FUNCTION_BLOCK PUBLIC ABSTRACT FB_HMI_PROVIDER_BASE IMPLEMENTS ITF_HMI_PROVIDER
VAR_INPUT
END_VAR
VAR_OUTPUT
END_VAR
VAR
	eProvider	: E_HMI_PROVIDER;
	
	stItfHmiIn	: REFERENCE TO ST_HMI_IN;
	stItfHmiOut	: REFERENCE TO ST_HMI_OUT;
	
	bRequestManualControl,
	bRequestRecipeMgmt,
	bRequestSettingMgmt,
	bRequestUserMgmt,
	bMute		: BOOL;
END_VAR

PROPERTY ItfHmiIn : REFERENCE TO ST_HMI_IN
GET
ItfHmiIn REF= stItfHmiIn;
END_GET
END_PROPERTY

PROPERTY ItfHmiOut : REFERENCE TO ST_HMI_OUT
GET
ItfHmiOut REF= stItfHmiOut;
END_GET
END_PROPERTY

METHOD PUBLIC M_Init : BOOL
VAR_INPUT
END_VAR
P_HMI_Controller.M_RegisterProvider(THIS^);
M_Init := TRUE;
END_METHOD

(* reset*)
METHOD M_Reset : BOOL
stItfHmiIn.stSpecial.stButton_LedTest.bClick := FALSE;
END_METHOD

METHOD M_Run : BOOL
VAR
	msg : STRING;
END_VAR
IF NOT RefsValid THEN
	msg := CONCAT('HMI provider ref error, provider: ', TO_STRING(eProvider));
	Services.fbEventHandler.Select(TC_Events.SystemEventClass.ErrorEvent).ArgSetString(msg).Raise();
	RETURN;
END_IF

M_Run := TRUE;
END_METHOD

METHOD M_SetReferencesBase : BOOL
VAR_IN_OUT
	stHmiPrvIn	: ST_HMI_IN;
	stHmiPrvOut	: ST_HMI_OUT;
END_VAR
stItfHmiIn REF= stHmiPrvIn;
stItfHmiOut REF= stHmiPrvOut;
stItfHmiOut.stCommon REF= HMI.stHmi.stOut.stCommon; // same common out 4 all HMI provider, in order to save memory
M_SetReferencesBase := TRUE;
END_METHOD

PROPERTY Mute : bool
GET
Mute := bMute;
END_GET
END_PROPERTY

{attribute 'monitoring' := 'call'}
PROPERTY Provider : E_HMI_PROVIDER
GET
Provider := eProvider;
END_GET
END_PROPERTY

{attribute 'monitoring' := 'call'}
PROPERTY RefsValid : bool
GET
RefsValid := __ISVALIDREF (stItfHmiIn) AND_THEN
			 __ISVALIDREF (stItfHmiOut);
END_GET
END_PROPERTY

(* HMI control request (Bedienhoheit)
	set ti true, on any control request from the HMI provider (e.g.: watch IN struct)
	reset will be done by HMI controller, on other provider request  *)
{attribute 'monitoring':='call'}
PROPERTY RequestManualControl : BOOL
GET
RequestManualControl := bRequestManualControl;
END_GET
SET
bRequestManualControl := RequestManualControl;
END_SET
END_PROPERTY

(* HMI recipe control request (Bedienhoheit)  *)
{attribute 'monitoring':='call'}
PROPERTY RequestRecipeMgmt : BOOL
GET
RequestRecipeMgmt := bRequestRecipeMgmt;
END_GET
SET
bRequestRecipeMgmt := RequestRecipeMgmt;
END_SET
END_PROPERTY

(* HMI recipe control request (Bedienhoheit)  *)
{attribute 'monitoring':='call'}
PROPERTY RequestSettingMgmt : BOOL
GET
RequestSettingMgmt := bRequestSettingMgmt;
END_GET
SET
bRequestSettingMgmt := RequestSettingMgmt;
END_SET
END_PROPERTY

(* HMI user management control request (Bedienhoheit)  *)
{attribute 'monitoring':='call'}
PROPERTY RequestUserMgmt : BOOL
GET
RequestUserMgmt := bRequestUserMgmt;
END_GET
SET
bRequestUserMgmt := RequestUserMgmt;
END_SET
END_PROPERTY

END_FUNCTION_BLOCK

(* stored: Version 1.1.0.1
   POU FB_HMI_PROVIDER_BASE: Id {eb3b13ab-0697-40da-bd0e-8c1192b792bf}, SpecialFunc None
   Folder Methods: Id {4371ce8a-2be0-45a5-b48d-5497abc89aa2}
   Folder Properties: Id {19560e8a-6f53-4c5f-9456-58c06c8dabc4}
   Property ItfHmiIn: Id {8b135c92-9e5a-4ab2-b5fd-c25b1745d8d6}
   Get Get: Id {b891f3cc-a6f7-4957-ae98-f890cff48ca7}
   Property ItfHmiOut: Id {f4aa119e-6666-4149-af84-fef70564cbdf}
   Get Get: Id {5866c261-7b3f-4b0d-aa28-bba29b67a015}
   Method M_Init: Id {a4774064-60f7-454a-9e5f-5d827598134b}
   Method M_Reset: Id {9562efb1-6147-494f-83ee-a33594a3d96d}
   Method M_Run: Id {b599e4b7-dc6c-4993-b682-12468ee2a04f}
   Method M_SetReferencesBase: Id {0ff96172-e091-4d24-a480-742ad33456ff}
   Property Mute: Id {d75ff4f9-7601-4c81-9ef8-8ea6f6cf481f}
   Get Get: Id {d487fae3-837d-49a4-a40b-538d2339b2b5}
   Property Provider: Id {4ea6dd9c-1e46-48cf-be6e-7e59c2bf8b4d}
   Get Get: Id {8e5f494e-dd2f-43ab-8cfe-54151534583c}
   Property RefsValid: Id {8239054e-eeb0-47bf-9ce3-424e994992d4}
   Get Get: Id {bd066d3e-c968-4cc6-971a-201385bd1eef}
   Property RequestManualControl: Id {8f49d3cd-a26b-4750-b17d-cf255f6e839f}
   Get Get: Id {2e9b6ac1-1488-4140-a4b9-387b159c447c}
   Set Set: Id {c1b4e7f8-fd62-4efa-9b5d-72bff59ff4de}
   Property RequestRecipeMgmt: Id {7523044a-7388-4ac4-9d7c-e75c3cc23c4a}
   Get Get: Id {6669e8ec-3ce8-4ea2-8125-f60aa98d485c}
   Set Set: Id {d1660c92-acd3-4443-bd97-8d4e7c8fc4e7}
   Property RequestSettingMgmt: Id {9a40c98e-d4fe-46f5-b48e-e1c994c8d2d8}
   Get Get: Id {2c21a599-0dd5-4e7e-921a-cfcbe6a2a409}
   Set Set: Id {366428d0-25e6-4864-b0d6-e762050abc23}
   Property RequestUserMgmt: Id {111e378e-f6b8-4f1e-9276-f72b13017db8}
   Get Get: Id {3d90ba8b-7e99-47d1-9ac4-f059769e3ae6}
   Set Set: Id {13f9f8c7-c3c4-4344-a3c8-1afcd5e648f4} *)
